//Cases to handle the automatic setup of the checker board
CASE caseState OF
	//Initialization of all the variables 
	000:
		IF (GVL.boardIsSetup = TRUE) THEN
			currentChecker :=0;
			currentStack := 0;
			currentStackPosition := 0;
			caseState := 010;
		END_IF
	//Moving Z axis up to start move to first stack	
	010:
		movePiece.zPos := zUp;
		caseState := 020;
	//Execute of the above move	
	020:
		movePiece.ExecuteMove := TRUE;
		caseState := 030;
	//Check to make sure above move finished
	030:
		IF (movePiece.MoveDone) THEN
			caseState := 190;
			movePiece.ExecuteMove := FALSE;
		END_IF
		
	//Input of the x and y coordinates of the stack that is currently getting picked from
	040:
		IF (currentStack < 3 ) THEN
			movePiece.xPos := xStackOffset + (xStackDistance * currentStack);
			movePiece.yPos := yStackOffset + (yStackDistance * currentStack);		
			movePiece.zPos := zUp;
			caseState := 050;
		END_IF
		
		IF (currentStack >=3 AND currentStack < 6 ) THEN
			movePiece.xPos := xStackOffset + (xStackDistance * currentStack);
			movePiece.yPos := yStackOffset + (yStackDistance * currentStack);		
			movePiece.zPos := zUp;
			caseState := 050;			
		END_IF
	//Execution of the move to the current stack being picked from	
	050:
		movePiece.ExecuteMove := TRUE;
		caseState := 060;
	//Check to make sure the execution of the move to the first stack was completed
	060:
		IF (movePiece.MoveDone) THEN
			caseState := 070;
			movePiece.ExecuteMove := FALSE;
		END_IF
	//Moving Z axis down to pick up the current checker and incrementing the stack position 
	070:
		movePiece.zPos := zDown - pieceOffset * ( 4 - currentStackPosition);
		currentStackPosition := currentStackPosition +1;
		IF (currentStackPosition = 5) THEN
			currentStackPosition := 0;
			currentStack := currentStack + 1;
			IF(currentStack = 2 OR currentStack = 5) THEN 
				currentStackPosition := 3;
			END_IF
		END_IF
		caseState := 080;
	//Execution of the z axis move downward to pick up current checker from current stack
	080:
		movePiece.ExecuteMove := TRUE;
		caseState := 090;
	//Check to make sure that the z axis move was properly executed, and closing of the gripper and delay to make sure that the gripper grabs the checker
	090:
		IF (movePiece.MoveDone) THEN
			caseState := 100;
			movePiece.ExecuteMove := FALSE;
			gripperMove := TRUE;
			wait.startTimer := TRUE;
		END_IF
	//Waiting for the timer to finish and then reinitializing it as false, as well as moving the z axis back up to move to the proper checker space
	100:
		IF (wait.done) THEN
			wait.startTimer := FALSE;
			gripperMove := FALSE;
			movePiece.zPos := zUp;
			caseState := 110;
		END_IF
	//Execution of the Z-axis move upwards to start move to proper board location 	
	110:
		movePiece.ExecuteMove := TRUE;
		caseState := 120;
	//Check to make sure that the above move is completed
	120: 
		IF (movePiece.MoveDone) THEN
			caseState := 130;
			movePiece.ExecuteMove := FALSE;
		END_IF
	//Input of x and y coordinates to proper checker board location depending on the color of the checker and the current check being placed
	130:
		IF (currentChecker < 12) THEN
			movePiece.xPos := xBoardOffset + (GVL.pieces[0,currentChecker].startingLocation[0] * spaceOffset); 
			movePiece.yPos := yboardOffset + (GVL.pieces[0,CurrentChecker].startingLocation[1] * spaceOffseT);
			currentChecker := currentChecker+1;
			caseState := 140;
		END_IF
		
		IF (currentChecker >= 12 AND currentChecker < 24) THEN
			movePiece.xPos := xBoardOffset + (GVL.pieces[1,currentChecker].startingLocation[0] *spaceOffset); 
			movePiece.yPos := yboardOffset + (GVL.pieces[1,CurrentChecker].startingLocation[1] *spaceOffseT);
			currentChecker := currentChecker+1;
			caseState :=140;
		END_IF
	//Execution of the above move to place checker on the proper board square	
	140:
		movePiece.ExecuteMove := TRUE;
		caseState := 150;
	//Check to make sure that the above move was completed	
	150:
		IF (movePiece.MoveDone) THEN;
			caseState := 160 ;
			movePiece.ExecuteMove := FALSE;
		END_IF
	//Move Z axis down to board level to prepare to drop it off	
	160:
		movePiece.zPos := zDown;
		caseState := 170;
	//Execution of the downward movement of the z axis to drop off the checker
	170:
		movePiece.ExecuteMove := TRUE;
		caseState := 180;
	//Check to make sure z axis moved, and opening the grippers to drop the current checker on the board square
	180:
		IF (movePiece.MoveDone) THEN
			caseState := 190;
			movePiece.ExecuteMove := FALSE;
			gripperMove := TRUE;
			wait.startTimer := TRUE;
		END_IF
	//Re-initializing the timer function and reseting the z axis above the board
	190:
		IF (wait.done) THEN
			wait.startTimer := FALSE;
			gripperMove := FALSE;
			movePiece.zPos := zUp;
			caseState := 020;
		END_IF
		
		IF (currentChecker = 23) THEN
			caseState := 200;
		END_IF
	//Case to hold program until the board is called to be reset
	200:
		IF (gameReset = TRUE) THEN
			caseState := 000;
		END_IF
END_CASE

movePiece(AxisGroup := XYZ);
wait();

END_PROGRAM

// CODESYS_SoftMotion_Win_V3/Application/GameplayFunctions/movePiece
FUNCTION movePiece : Piece
VAR_INPUT
	currentPiece : Piece;
	spaceX : INT; // space that you the user wants to move to
	spaceY : INT; // space that the user wants to move to
END_VAR
VAR
	spaceTranslation : ARRAY [0..1] OF INT; // small numbers (0-7) that indicate how many spaces a piece needs to be moved
	sizeOfMoveX : INT := 50;
	sizeOfMoveY : INT := -50;
END_VAR

// DOESN'T DO ANYTHING, DEPRECATE


IF(currentPiece.validMoveArr[spaceX, spaceY]) THEN
	
	// Tells you how many spaces you need to move
	spaceTranslation[0] := spaceX - currentPiece.currentLocation[0];
	spaceTranslation[1] := spaceY - currentPiece.currentLocation[1];

	// Converts spaces needed to move into pixels needed to move
	currentPiece.translatedLocation[0] := spaceTranslation[0] * sizeOfMoveX;
	currentPiece.translatedLocation[1] := spaceTranslation[1] * sizeOfMoveY;
	
	// sets old location to the current location
	currentPiece.oldLocation[0] := currentPiece.currentLocation[0];
	currentPiece.oldLocation[1] := currentPiece.currentLocation[1];
	
	// updates the current location
	currentPiece.currentLocation[0] := spaceX;
	currentPiece.currentLocation[1] := spaceY;
	
END_IF

movePiece := currentPiece;
currentPiece.isSelected := FALSE;

RETURN;

END_FUNCTION

// CODESYS_SoftMotion_Win_V3/Application/GameplayFunctions/HMISequence
PROGRAM HMISequence
VAR
END_VAR

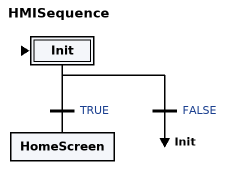
INITIAL_STEP Init:
END_STEP
TRANSITION FROM Init TO HomeScreen
    := TRUE;
END_TRANSITION
TRANSITION FROM Init TO Init
    := FALSE;
END_TRANSITION
STEP HomeScreen:
END_STEP

END_PROGRAM

// CODESYS_SoftMotion_Win_V3/Application/GameplayFunctions/Init
PROGRAM Init
VAR
END_VAR

END_PROGRAM

// CODESYS_SoftMotion_Win_V3/Application/GameplayFunctions/JumpPieces
PROGRAM JumpPieces
VAR
	i : INT;
	selectedPieceColor : INT;
	selectedPieceIndex : INT;
END_VAR

END_PROGRAM

// CODESYS_SoftMotion_Win_V3/Application/GameplayFunctions/pieceSelect
FUNCTION pieceSelect : ARRAY[0..1,0..11] OF Piece;
VAR_INPUT
	pieces : ARRAY[0..1,0..11] OF Piece;
	selectedPieceValidMoveArr : ARRAY[0..7,0..7] OF BOOL;
END_VAR
VAR
	i :INT;
END_VAR

FOR i := 0 TO 11 DO
	pieces[0,i].isSelected := FALSE;
	pieces[1,i].isSelected := FALSE;
END_FOR

selectedPieceValidMoveArr := pieces[0,10].validMoveArr;
pieceSelect := pieces;

END_FUNCTION

// CODESYS_SoftMotion_Win_V3/Application/GameplayFunctions/placePiece
FUNCTION placePiece : ARRAY [0..1] OF INT

VAR_INPUT
	isBlack : BOOL;
	pieceNum : INT;
END_VAR
VAR
	x : INT;
	y : INT;
	temp : INT;
END_VAR

// Set up for black
IF(isBlack) THEN
	y := pieceNum / 4;
	x := ((2 * pieceNum) MOD 8) + (y MOD 2);
// Setup for red
ELSE
	temp := pieceNum / 4;
	y := temp + 5;
	x := (((2 * pieceNum) MOD 8) + (temp MOD 2)) + 1;
	IF(x >= 8) THEN
		x := 0;
	END_IF
END_IF

placePiece[0] := x;
placePiece[1] := y;

RETURN;

END_FUNCTION

// CODESYS_SoftMotion_Win_V3/Application/GameplayFunctions/ProgramFlow
PROGRAM ProgramFlow
VAR
	PlayGame: BOOL;
END_VAR
// where we displace player move options?

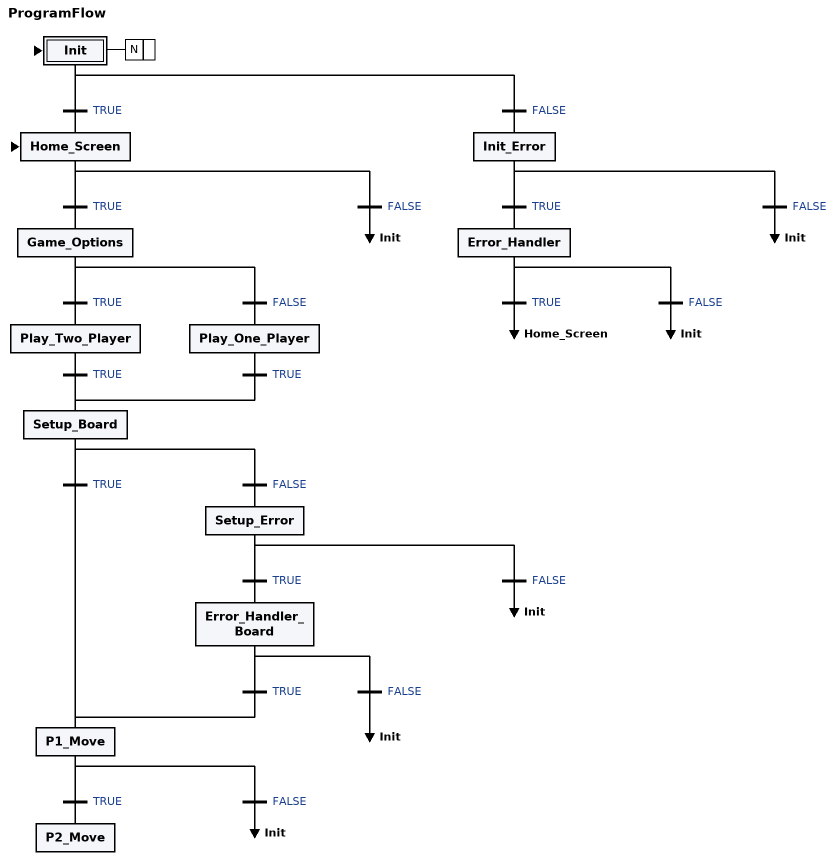
INITIAL_STEP Init:
    // ???(N);
END_STEP
TRANSITION FROM Init TO Home_Screen
    := TRUE;
END_TRANSITION
TRANSITION FROM Init TO Init_Error
    := FALSE;
END_TRANSITION
STEP Init_Error:
END_STEP
TRANSITION FROM Init_Error TO Error_Handler
    := TRUE;
END_TRANSITION
STEP Error_Handler:
END_STEP
TRANSITION FROM Error_Handler TO Home_Screen
    := TRUE;
END_TRANSITION
TRANSITION FROM Error_Handler TO Init
    := FALSE;
END_TRANSITION
TRANSITION FROM Init_Error TO Init
    := FALSE;
END_TRANSITION
STEP Home_Screen:
END_STEP
TRANSITION FROM Home_Screen TO Game_Options
    := TRUE;
END_TRANSITION
TRANSITION FROM Home_Screen TO Init
    := FALSE;
END_TRANSITION
STEP Game_Options:
END_STEP
TRANSITION FROM Game_Options TO Play_Two_Player
    := TRUE;
END_TRANSITION
STEP Play_Two_Player:
END_STEP
TRANSITION FROM Play_Two_Player TO Setup_Board
    := TRUE;
END_TRANSITION
TRANSITION FROM Game_Options TO Play_One_Player
    := FALSE;
END_TRANSITION
STEP Play_One_Player:
END_STEP
TRANSITION FROM Play_One_Player TO Setup_Board
    := TRUE;
END_TRANSITION
STEP Setup_Board:
END_STEP
TRANSITION FROM Setup_Board TO P1_Move
    := TRUE;
END_TRANSITION
TRANSITION FROM Setup_Board TO Setup_Error
    := FALSE;
END_TRANSITION
STEP Setup_Error:
END_STEP
TRANSITION FROM Setup_Error TO Error_Handler_Board
    := TRUE;
END_TRANSITION
TRANSITION FROM Setup_Error TO Init
    := FALSE;
END_TRANSITION
STEP Error_Handler_Board:
END_STEP
TRANSITION FROM Error_Handler_Board TO P1_Move
    := TRUE;
END_TRANSITION
TRANSITION FROM Error_Handler_Board TO Init
    := FALSE;
END_TRANSITION
STEP P1_Move:
END_STEP
TRANSITION FROM P1_Move TO P2_Move
    := TRUE;
END_TRANSITION
TRANSITION FROM P1_Move TO Init
    := FALSE;
END_TRANSITION
STEP P2_Move:
END_STEP

END_PROGRAM

// CODESYS_SoftMotion_Win_V3/Application/GameplayFunctions/MoveHome
PROGRAM MoveHome
VAR
	moveToHome : MovePieceMotion;
	caseState: INT;
END_VAR

CASE caseState OF
	
000: 
	IF(GVL.homeAxes)THEN
		moveToHome.xPos := 0;
		moveToHome.yPos := 0;
		moveToHome.zPos := 0;
		caseState := 010;
	END_IF

010:
	moveToHome.ExecuteMove := TRUE;
	caseState := 020;

020:
	IF(moveToHome.MoveDone)THEN
		moveToHome.ExecuteMove := FALSE;
		caseState := 000;
		GVL.homeAxes := FALSE;
	END_IF
	
	
END_CASE

moveToHome();

END_PROGRAM

// CODESYS_SoftMotion_Win_V3/Application/GameplayFunctions/SetupFromStart
PROGRAM SetupFromStart
VAR
END_VAR

END_PROGRAM

// CODESYS_SoftMotion_Win_V3/Application/ArrayMove
FUNCTION_BLOCK ArrayMove
VAR_INPUT
	//TestArray: ARRAY [1..20] OF INT := [1,2,3,4,5,6,7,8,9,10,11,12,13,14,15,16,17,18,19,20];
	i: INT ; 
END_VAR
VAR_OUTPUT
END_VAR
VAR
	Done : BOOL;
END_VAR

IF(NOT Done) THEN	
	FOR i:= 20 TO 2 BY -1 DO 
		PersistentVars.MyArray[i]:= PersistentVars.MyArray [i-1];
	END_FOR
	PersistentVars.MyArray[1].Names := GlobalVars.winnerName;
	PersistentVars.MyArray[1].Moves := GlobalVars.winnerMoves;
	Done := TRUE;
END_IF

END_FUNCTION_BLOCK

// CODESYS_SoftMotion_Win_V3/Application/GameplayFunctions/TestMyArray
PROGRAM TestMyArray
VAR
	k : INT ; 
	arrayTest : ArrayMove;
END_VAR

arrayTest();
//k := ArrayMove.TestArray[2];

END_PROGRAM

// CODESYS_SoftMotion_Win_V3/Application/Export/GetHeaderString
FUNCTION GetHeaderString : STRING[255]
VAR_INPUT
END_VAR
VAR
	msg: STRING[255];
	seperator: STRING;
	eol:String;
	strTemp0 : STRING[255];
	strTemp1 : STRING[255];
	

END_VAR

eol := WORD_AS_STRING(16#0A0D, FALSE);
seperator := ',';

strTemp0 := Concat(Concat(	'Winners', 
						 seperator), 
						    'Moves');




GetHeaderString := Concat(Concat(Concat(Concat(	'TimeStamp', 
														seperator),
														strTemp0), 
														seperator),
						     								eol);

END_FUNCTION

// CODESYS_SoftMotion_Win_V3/Application/Export/GetLogMsgString
FUNCTION GetLogMsgString : STRING[255]
VAR_INPUT
END_VAR
VAR
	msg: STRING[255];
	seperator: STRING;
	eol:String;
	
	DataPrep: STRING[255];
	
	
END_VAR

eol := WORD_AS_STRING(16#0A0D, FALSE);
seperator := ',';


DataPrep := Concat(Concat(  PersistentVars.MyArray[1].Names,
                                                  seperator),
            INT_TO_STRING(PersistentVars.MyArray[1].Moves));
																												



GetLogMsgString := Concat(Concat(Concat(Concat(	GetTimeStampString(),
														seperator),
														DataPrep), 
														seperator),
															eol);

END_FUNCTION

// CODESYS_SoftMotion_Win_V3/Application/Export/GetTimeStampString
FUNCTION GetTimeStampString : STRING
VAR_INPUT
END_VAR
VAR
	TimeStamp : SysTime;
	StructTimeStamp : SysTimeDate;
	Result : RTS_IEC_RESULT;
	StrDate : STRING;
	StrTime : STRING;
	

END_VAR

Result := systimertc.SysTimeRtcHighResGet(pTimestamp := TimeStamp);

Result := systimertc.SysTimeRtcConvertHighResToLocal(pTimeStamp:=TimeStamp, pDate:=StructTimeStamp);

StrDate := UINT_TO_STRING(StructTimeStamp.wYear);
IF StructTimeStamp.wMonth < 10 THEN 
	StrDate := Concat(Concat(StrDate, '0') , UINT_TO_STRING(StructTimeStamp.wMonth));
ELSE
	StrDate := Concat(StrDate , UINT_TO_STRING(StructTimeStamp.wMonth));
END_IF

IF StructTimeStamp.wDay < 10 THEN 
	StrDate := Concat(Concat(StrDate , '0') , UINT_TO_STRING(StructTimeStamp.wDay));
ELSE
	StrDate := Concat(StrDate , UINT_TO_STRING(StructTimeStamp.wDay));
END_IF


IF StructTimeStamp.wHour < 10 THEN 
	StrTime := Concat(Concat('0' , UINT_TO_STRING(StructTimeStamp.wHour)) , ':');
ELSE
	StrTime := Concat(UINT_TO_STRING(StructTimeStamp.wHour) , ':');
END_IF

IF StructTimeStamp.wMinute < 10 THEN 
	StrTime := Concat(Concat(Concat(StrTime , '0') , UINT_TO_STRING(StructTimeStamp.wMinute)), ':');
ELSE
	StrTime := Concat(Concat(StrTime , UINT_TO_STRING(StructTimeStamp.wMinute)), ':');
END_IF

IF StructTimeStamp.wSecond < 10 THEN 
	StrTime := Concat(Concat(Concat(StrTime , '0') , UINT_TO_STRING(StructTimeStamp.wSecond)) , '.');
ELSE
	StrTime := Concat(Concat(StrTime , UINT_TO_STRING(StructTimeStamp.wSecond)) , '.');
END_IF

IF StructTimeStamp.wMilliseconds < 10 THEN 
	StrTime := Concat(Concat(StrTime , '00') , UINT_TO_STRING(StructTimeStamp.wMilliseconds));
ELSE
	IF StructTimeStamp.wMilliseconds < 100 THEN 
		StrTime := Concat(Concat(StrTime , '0') , UINT_TO_STRING(StructTimeStamp.wMilliseconds));
	ELSE
		StrTime := Concat(StrTime , UINT_TO_STRING(StructTimeStamp.wMilliseconds));
	END_IF
END_IF

//GetTimeStampString := Concat(Concat(strDate , '-'), strTime);
GetTimeStampString := strTime;

END_FUNCTION

// CODESYS_SoftMotion_Win_V3/Application/Export/LogWinnerNames
PROGRAM LogWinnerNames
VAR
	strMsg: STRING[255];
	iStatus : INT := 0;
	LogIndex :DINT := 0;
	LogMsg : ARRAY [1..200] OF STRING[255];
	LogType : STRING;
	
	CycleTimeWarning: DWORD := 600;
	TotalSyncBufferAvgWarning: DINT := 125;
	CycleTimeError: DWORD := 900;
	TotalSyncBufferAvgError: DINT := 200;
	
	
	
END_VAR

VAR_INPUT
	bResetArray: BOOL;
END_VAR

IF bResetArray = TRUE THEN
	LogIndex := 0;
END_IF




CASE iStatus OF
	

0:	//Log Data
	LogIndex := LogIndex + 1;
	
	LogMsg[LogIndex] :=  GetLogMsgString();
	
	iStatus := 2;

END_CASE

END_PROGRAM

// CODESYS_SoftMotion_Win_V3/Application/Export/Run_FileCopy
PROGRAM Run_FileCopy
VAR
	RunTest: Test_FileCopy;
END_VAR

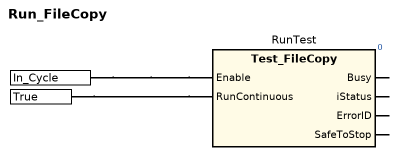
RunTest(Enable := In_Cycle, RunContinuous := True); // Test_FileCopy

END_PROGRAM

// CODESYS_SoftMotion_Win_V3/Application/Export/Test_FileCopy
FUNCTION_BLOCK Test_FileCopy
VAR_INPUT
	Enable: BOOL;
	RunContinuous:Bool := False;
END_VAR
VAR_OUTPUT
	Busy: BOOL;
	iStatus : INT := 0;
	ErrorID: INT;
	SafeToStop : Bool;
END_VAR
VAR
	OriginalFilePath : STRING := '/Hard disk/Backup/nk.bin';
	MemoryFilePath : STRING := '/nk.bin';
	USBFilePath : STRING := '/Hard disk2/nk.bin';
	DwellTime : TIME := T#15S;
	DoDwell : TON;
	
	Result1: SYSFILE.RTS_IEC_RESULT;
	Result2: SYSFILE.RTS_IEC_RESULT;

	BytesCopied: DWORD;
	SizeOriginal: DWORD;
	SizeMemory: DWORD;
	SizeUSB: DWORD;
END_VAR

IF Enable = FALSE and SafeToStop = True THEN
	iStatus := 0;
END_IF


CASE iStatus OF
	



0:  //Check Memory File Exist
	SafeToStop:=TRUE;
	SizeMemory := SysFileGetSize(MemoryFilePath, ADR(Result1));
	IF SizeMemory > 0 AND Result1 = Errors.ERR_OK THEN
		iStatus:=iStatus + 1;
	ELSE
		ErrorID := -1 * iStatus;  //Memory does not exist
		iStatus := 99;
	END_IF	

1:  //Check USB File Exist
	SafeToStop:=TRUE;
	SizeUSB := SysFileGetSize(USBFilePath, ADR(Result1));
	IF SizeUSB > 0 AND Result1 = Errors.ERR_OK THEN
		IF RunContinuous=TRUE THEN
			iStatus:=0;
		ELSE
			iStatus := 99;
		END_IF	
	ELSE
		ErrorID := -1 * iStatus;  //USB does not exist
		iStatus := 99;
	END_IF	
	
2:  // Copy to USBThumbdrive 
	SafeToStop:=FALSE;
	Result1:=SysFileCopy(USBFilePath,OriginalFilePath, ADR(BytesCopied));
	IF Result1=Errors.ERR_OK AND BytesCopied=SizeOriginal THEN
		iStatus:=iStatus + 1;
	ELSE
		ErrorID := -1 * iStatus;  //Copy to Memory Failed
		iStatus := 99;
	END_IF
	

3: //Got Error
	SafeToStop:=TRUE;
	Busy:=FALSE;
	
END_CASE

END_FUNCTION_BLOCK

// CODESYS_SoftMotion_Win_V3/Application/Visualizations/AreYouSure
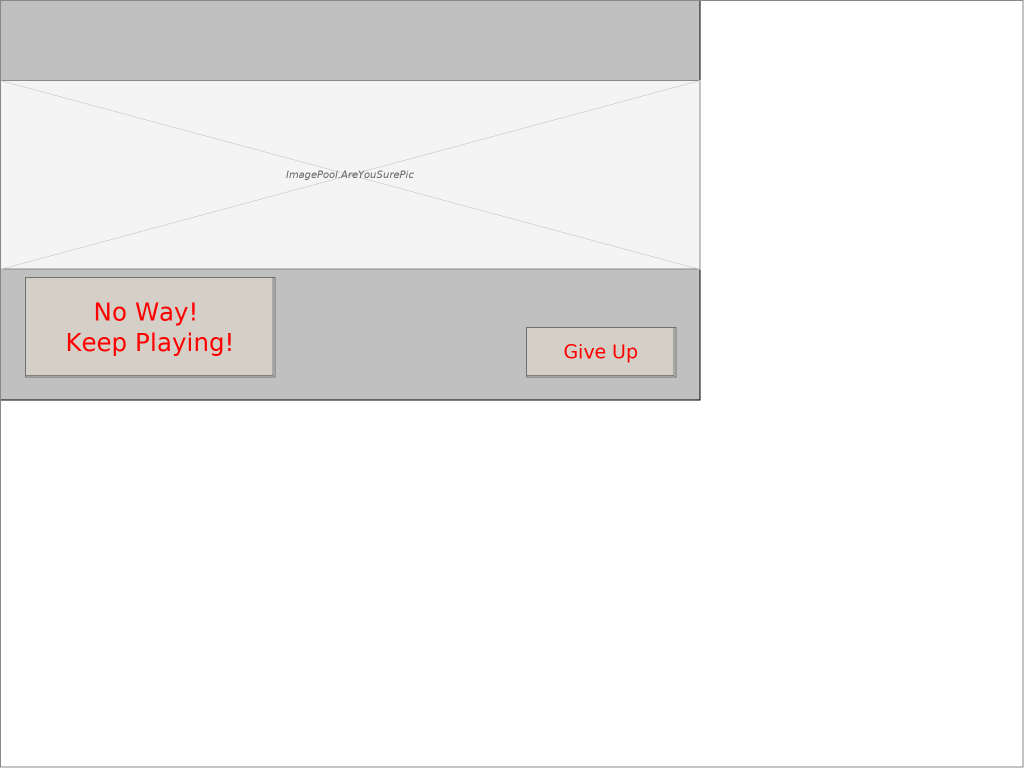
VISUALIZATION AreYouSure  // 1024x768
    Rectangle (0,0 700x400)
    Image (0,80 700x189), image: ImagePool.AreYouSurePic
    Button (25,277 250x100), "No Way! Keep Playing!"
        OnMouseClick:  Dialog=AreYouSure, Result=OK, NumpadKeypadSet=True
    Button (526,327 150x50), "Give Up"
        OnMouseClick:  Dialog=AreYouSure, Result=OK, NumpadKeypadSet=True
        OnMouseClick:  Assign=MainView, Type=Assignment
END_VISUALIZATION

// CODESYS_SoftMotion_Win_V3/Application/Visualizations/ErrorVis
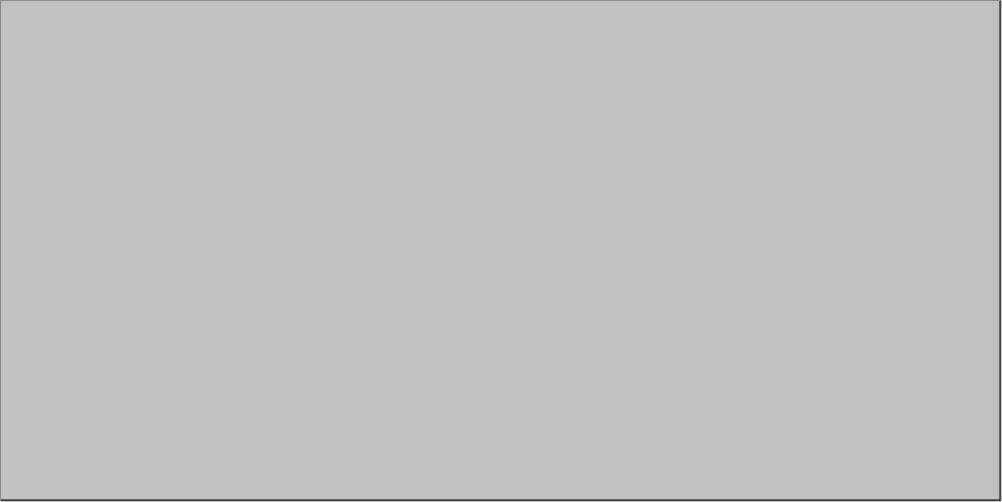
VISUALIZATION ErrorVis  // 1002x502
    Rectangle (0,0 1000x500)
END_VISUALIZATION

// CODESYS_SoftMotion_Win_V3/Application/Visualizations/JogVis
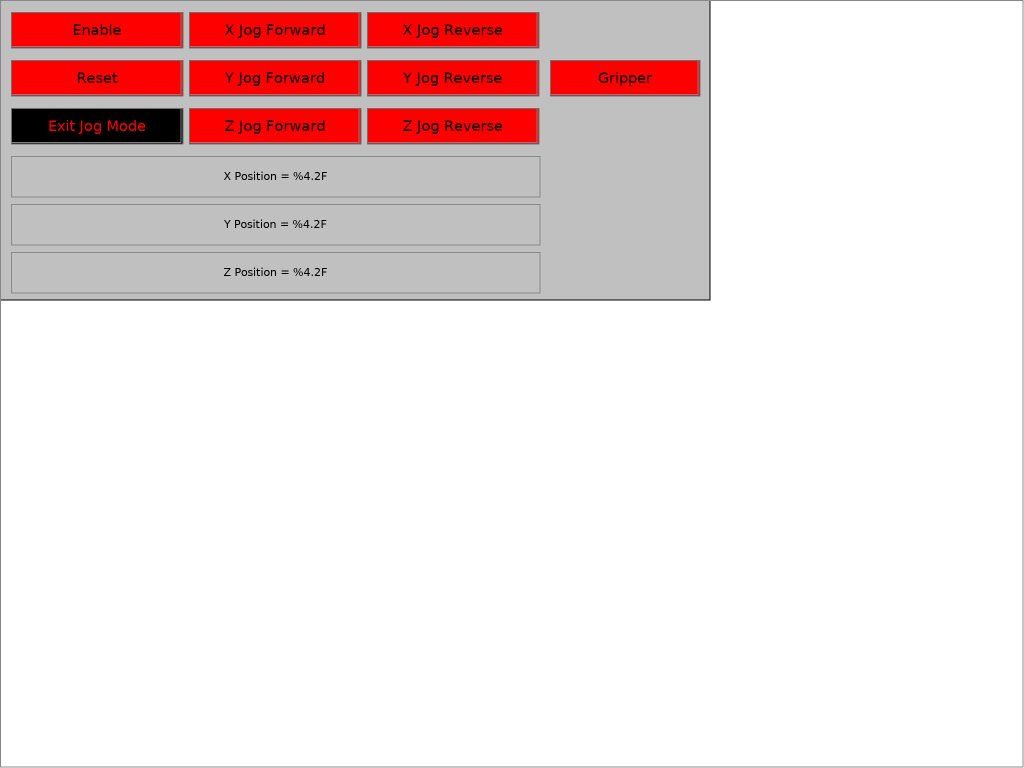
VISUALIZATION JogVis  // 1024x768
    Rectangle (0,0 710x300)
    Button (11,12 172x36), "Enable"
        OnMouseClick:  ToggleVariable=TestPower.Enable
        OnMouseClick: execute { GlobalVars.systemEnable := TRUE; }
    Button (189,12 172x36), "X Jog Forward"
        tap JogLogic.xJogFwdPressed
    Button (367,12 172x36), "X Jog Reverse"
        tap JogLogic.xJogRevPressed
    Button (189,60 172x36), "Y Jog Forward"
        tap JogLogic.yJogFwdPressed
    Button (367,60 172x36), "Y Jog Reverse"
        tap JogLogic.yJogRevPressed
    Button (11,60 172x36), "Reset"
        OnMouseClick: execute { TestPower.systemReset := TRUE; }
    Button (189,108 172x36), "Z Jog Forward"
        tap JogLogic.zJogFwdPressed
    Button (367,108 172x36), "Z Jog Reverse"
        tap JogLogic.zJogRevPressed
    Frame (11,156 529x41), "X Position = %4.2F", text variable: X.fActPosition
        shows SM3_Basic.LinDrive(m_Input_AXISREF := X)
    Frame (11,204 529x41), "Y Position = %4.2F", text variable: Y.fActPosition
        shows SM3_Basic.LinDrive(m_Input_AXISREF := Y)
    Frame (11,252 529x41), "Z Position = %4.2F", text variable: Z.fActPosition
        shows SM3_Basic.LinDrive(m_Input_AXISREF := Z)
    Button (11,108 172x36), "Exit Jog Mode"
        OnMouseClick:  Dialog=JogVis, Result=OK, NumpadKeypadSet=True
    Button (550,60 150x36), "Gripper"
        toggle GripperMove
END_VISUALIZATION

// CODESYS_SoftMotion_Win_V3/Application/Visualizations/GameView
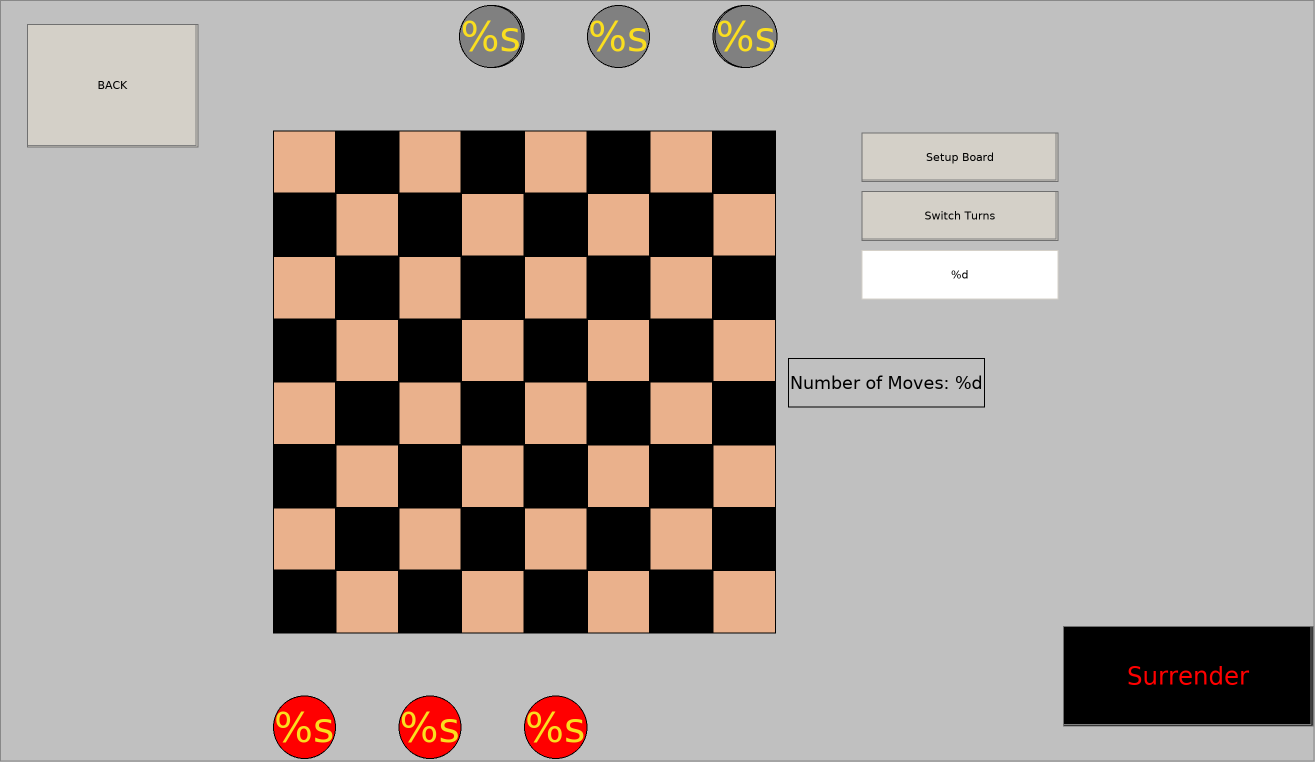
VISUALIZATION GameView  // 1315x762
    Frame (273,5 1005x755)
        shows Checkerboard()
    Button (27,24 171x123), "BACK"
        OnMouseClick:  Type=Previous
        OnMouseClick: execute { TestPower.GroupEnable := FALSE; }
    Button (1063,626 250x100), "Surrender"
        OnMouseClick:  Dialog=AreYouSure, OpenModal=True, OpenCentered=True
END_VISUALIZATION

// CODESYS_SoftMotion_Win_V3/Application/Visualizations/MainView
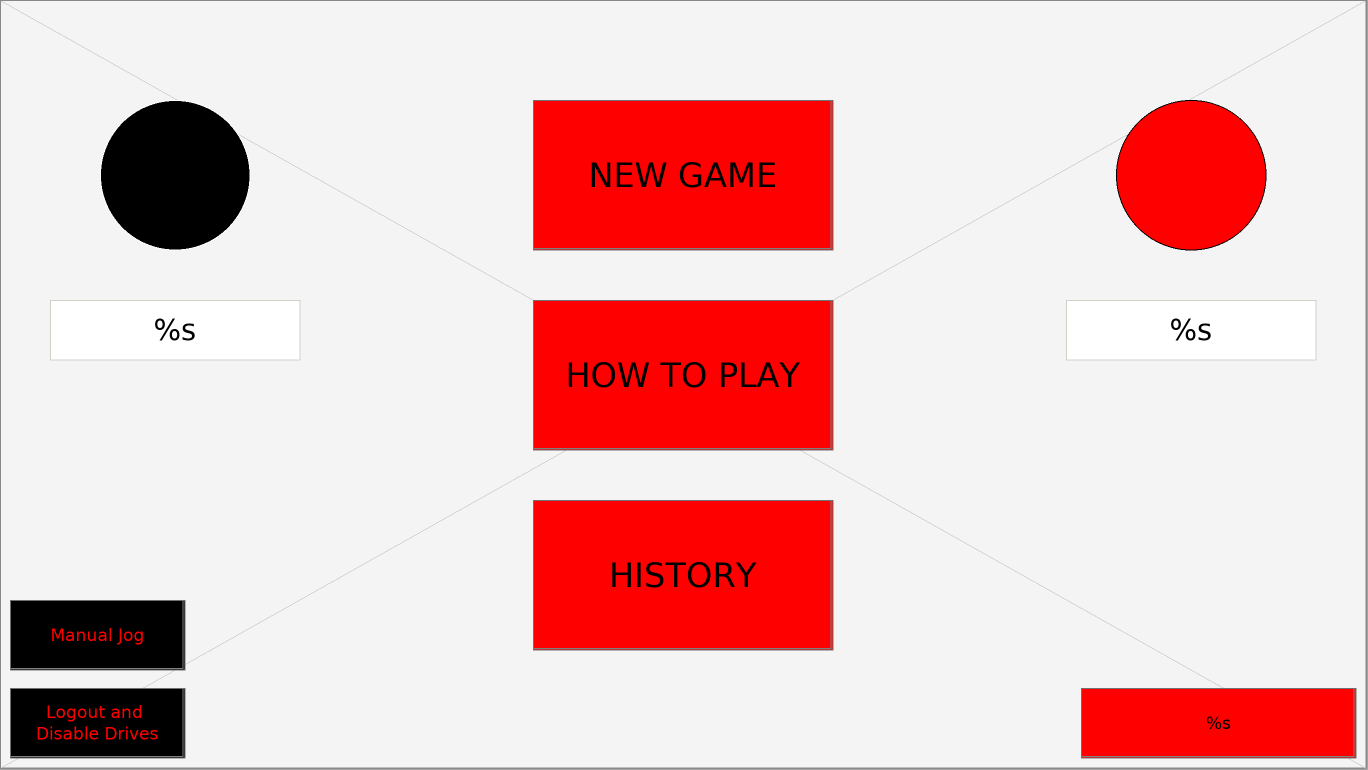
VISUALIZATION MainView  // 1368x770
    Image (0,0 1366x768), image: ImagePool.MedCheck_edited
    Ellipse (100,100 150x150), colour variable: GlobalVars.p1CheckerColor
    Ellipse (1116,100 150x150), colour variable: GlobalVars.p2CheckerColor
    Textfield (50,300 250x60), "%s", text variable: GlobalVars.p1Name
        OnMouseClick: write the text variable via Default
    Textfield (1066,300 250x60), "%s", text variable: GlobalVars.p2Name
        OnMouseClick: write the text variable via Default
    Button (533,100 300x150), "NEW GAME"
        OnMouseClick:  Assign=GameView, Type=Assignment
        OnMouseClick: execute { TestPower.GroupEnable := TRUE; }
    Button (533,300 300x150), "HOW TO PLAY"
        OnMouseClick:  Dialog=HowToPlay, OpenModal=True, OpenCentered=True
    Button (533,500 300x150), "HISTORY"
        OnMouseClick:  Dialog=History, OpenModal=True, OpenCentered=True
    Button (10,688 175x70), "Logout and Disable Drives"
        OnMouseClick:  Type=Logout
        OnMouseClick: execute { GlobalVars.systemEnable := FALSE; }
        OnMouseClick:  Assign=InitScreen, Type=Assignment
    Button (10,600 175x70), "Manual Jog"
        OnMouseClick:  Dialog=JogVis, OpenModal=True, OpenCentered=True, PositionX=0, PositionY=0
        OnMouseClick: execute { GlobalVars.systemEnable := TRUE; }
    Button (1081,688 275x70), "%s", text variable: GlobalVars.funnyText
        OnMouseClick: execute {
            GlobalVars.funnyCounter := GlobalVars.funnyCounter + 1;
            IF (GlobalVars.funnyCounter = 1) THEN
            	GlobalVars.funnyText := 'Stop it';
            ELSIF (GlobalVars.funnyCounter = 2) THEN
            	GlobalVars.funnyText := '.........';
            ELSIF (GlobalVars.funnyCounter = 3) THEN
            	GlobalVars.funnyText := 'How would you like it?';
            ELSIF (GlobalVars.funnyCounter = 4) THEN
            	GlobalVars.funnyText := 'Youre only wasting your time';
            ELSIF (GlobalVars.funnyCounter = 5) THEN
            	GlobalVars.funnyText := 'You win';
            ELSIF (GlobalVars.funnyCounter = 7) THEN
            	GlobalVars.funnyText := 'You dont give up easily';
            ELSIF (GlobalVars.funnyCounter = 8) THEN
            	GlobalVars.funnyText := 'Prize for your persistance';
            ELSIF (GlobalVars.funnyCounter = 9) THEN
            	GlobalVars.funnyText := 'lol';
            	VisuElems.CURRENTLANGUAGE := 'CowbellChinese';
            END_IF
        }
END_VISUALIZATION

// CODESYS_SoftMotion_Win_V3/Application/Visualizations/Congratulations
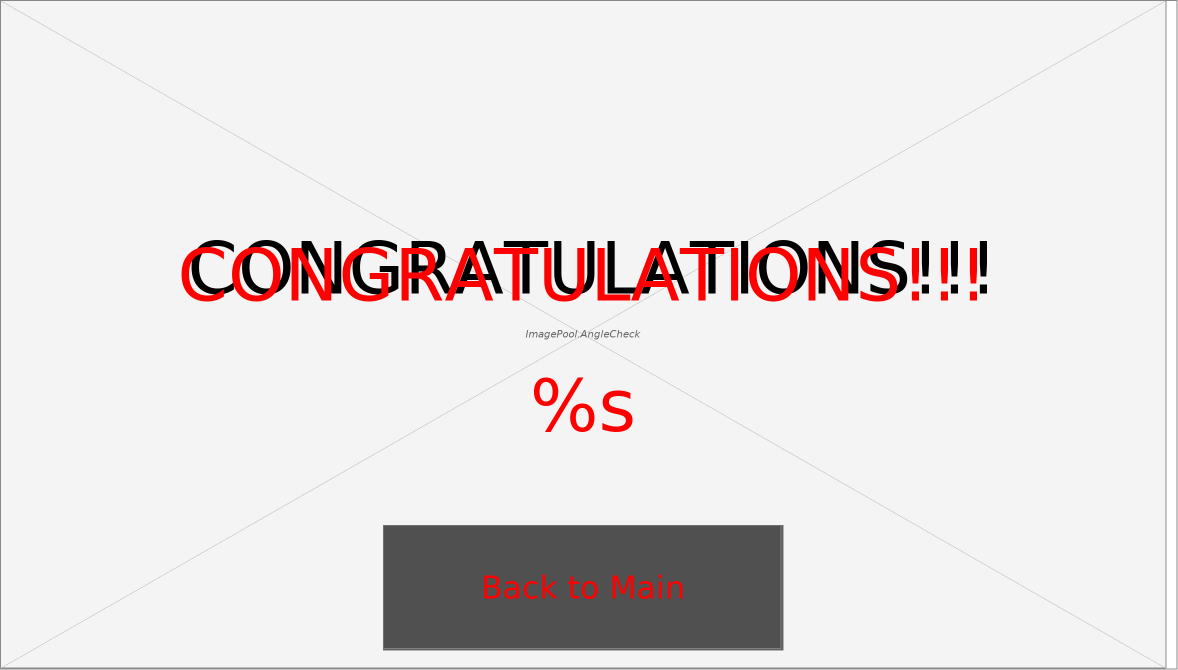
VISUALIZATION Congratulations  // 1178x670
    Image (0,0 1166x668), image: ImagePool.AngleCheck
    Rectangle (10,-7 1166x550), "CONGRATULATIONS!!!"
    Rectangle (0,0 1166x550), "CONGRATULATIONS!!!"
    Button (383,525 400x125), "Back to Main"
        OnMouseClick:  Assign=MainView, Type=Assignment
    Textfield (0,350 1166x111), "%s", text variable: GlobalVars.winnerName, colour variable: GlobalVars.p2CheckerColor
END_VISUALIZATION

// CODESYS_SoftMotion_Win_V3/Application/Visualizations/InitScreen
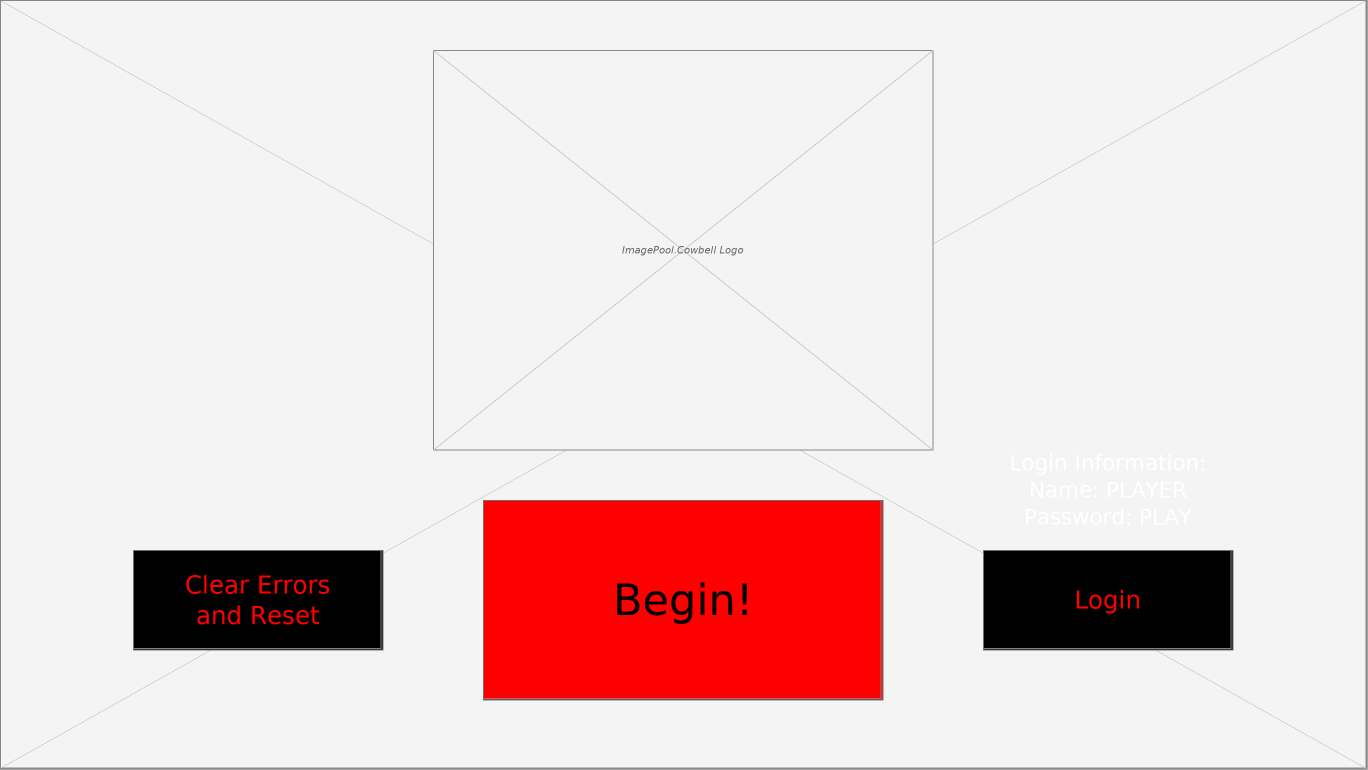
VISUALIZATION InitScreen  // 1368x770
    Image (0,0 1366x768), image: ImagePool.RedCheck
    Image (433,50 500x400), image: ImagePool.Cowbell Logo
    Button (483,500 400x200), "Begin!", text variable: GlobalVars.winnerName
        OnMouseClick:  Assign=MainView, Type=Assignment
        OnMouseClick: execute {
            TestPower.Enable := TRUE;
            JogLogic.startup := TRUE;
            // Run game setup code here
        }
    Button (983,550 250x100), "Login"
        OnMouseClick:  Type=Login
    Button (133,550 250x100), "Clear Errors and Reset"
        OnMouseClick: execute {
            VisuElems.CURRENTLANGUAGE := 'Default';
            JogLogic.startup := TRUE;
            // Any additional resets required to be done here
        }
        OnMouseClick:  Dialog=ErrorsCleared, OpenModal=True, OpenCentered=True
    Rectangle (983,440 250x100), "Login Information: Name: PLAYER Password: PLAY"
END_VISUALIZATION

// CODESYS_SoftMotion_Win_V3/Application/Visualizations/HowToPlay
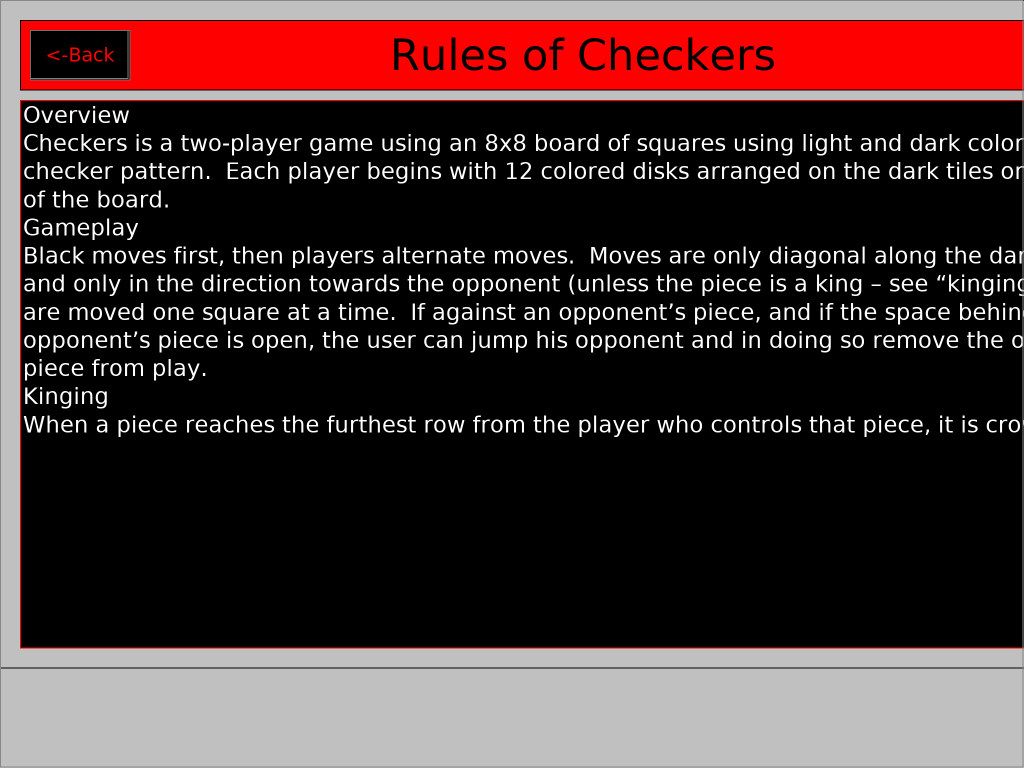
VISUALIZATION HowToPlay  // 1024x768
    Rectangle (0,0 1166x668)
    Textfield (20,100 1126x548), "Overview Checkers is a two-player game using an 8x8 board of squares using light and dark colors in a checker pattern. Each player begins with 12 colored disks arranged on the dark tiles on their side of the board. Gameplay Black moves first, then players alternate moves. Moves are only diagonal along the dark squares and only in the direction towards the opponent (unless the piece is a king – see “kinging”). Pieces are moved one square at a time. If against an opponent’s piece, and if the space behind the opponent’s piece is open, the user can jump his opponent and in doing so remove the opponent piece from play. Kinging When a piece reaches the furthest row from the player who controls that piece, it is crowned and becomes a king. One of the pieces which had been captured is placed on top of the king so that it is twice as high as a single piece. Kings may move both forward and backwards Winning A player wins the game when the opponent cannot make a move. In most cases, this is because all of the opponent's pieces have been captured, but it could also be because all of his pieces are blocked in."
    Textfield (20,20 1126x70), "Rules of Checkers"
    Button (30,30 100x50), "<-Back"
        OnMouseClick:  Dialog=HowToPlay, Result=OK, NumpadKeypadSet=True
END_VISUALIZATION

// CODESYS_SoftMotion_Win_V3/Application/Visualizations/ErrorsCleared
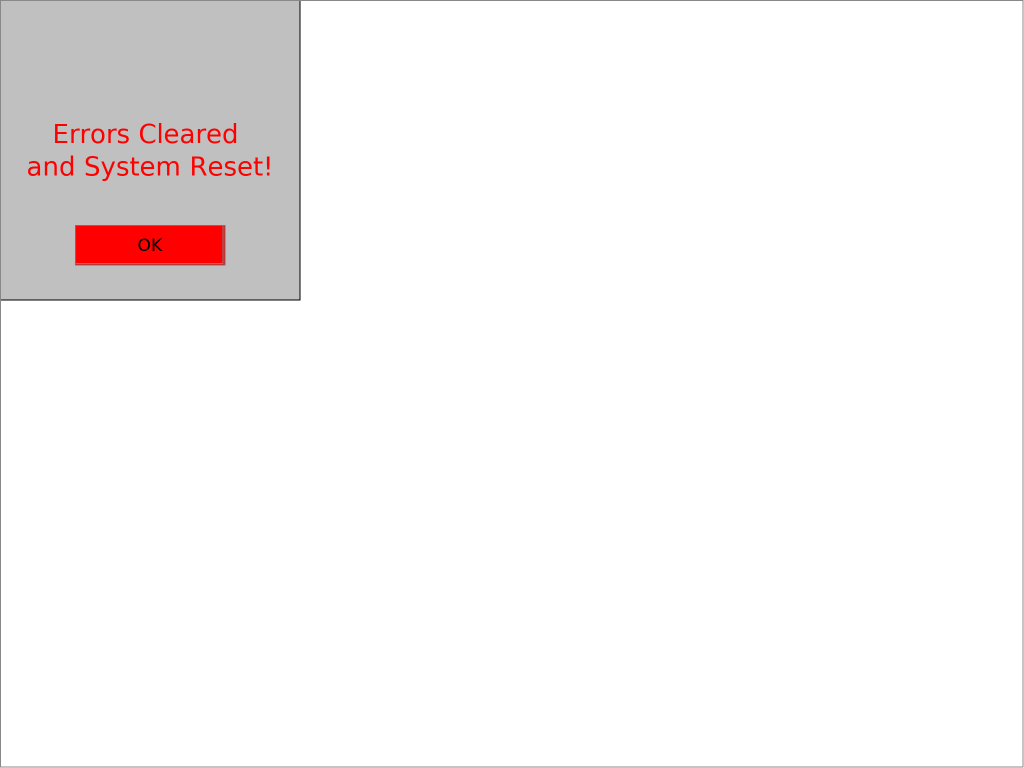
VISUALIZATION ErrorsCleared  // 1024x768
    Rectangle (0,0 300x300), "Errors Cleared and System Reset!"
    Button (75,225 150x40), "OK"
        OnMouseClick:  Dialog=ErrorsCleared, Result=OK, NumpadKeypadSet=True
END_VISUALIZATION

// CODESYS_SoftMotion_Win_V3/Application/Visualizations/Checkerboard
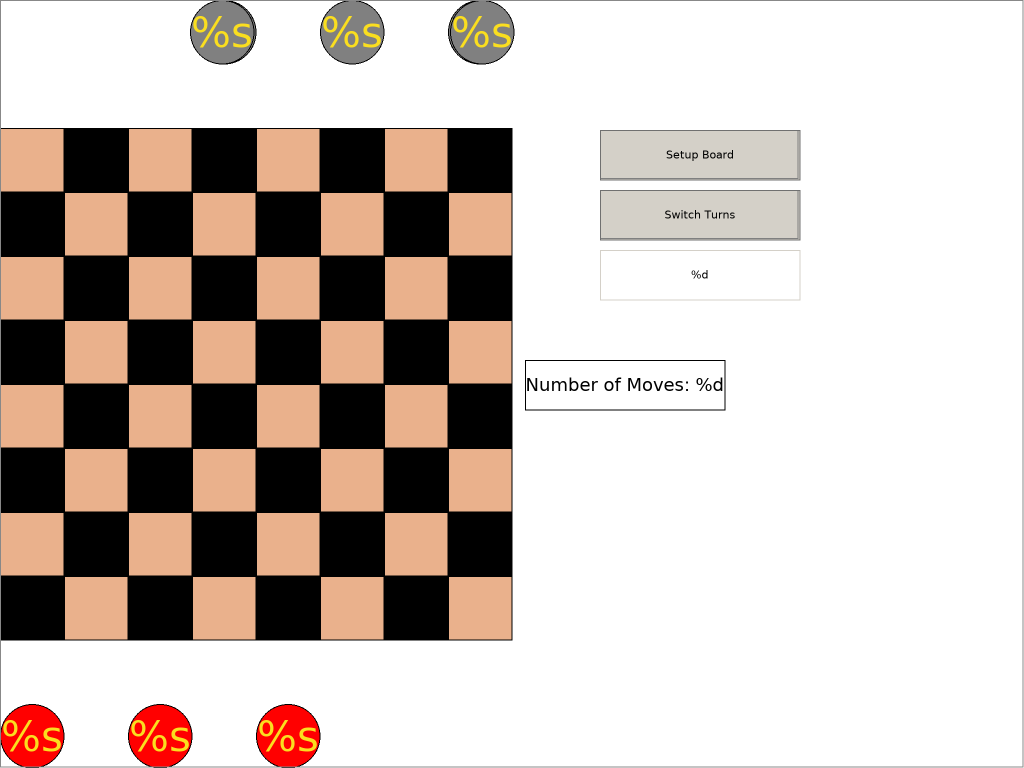
VISUALIZATION Checkerboard  // 1024x768
VAR_IN_OUT
	
END_VAR

VAR
	i : INT;
END_VAR
    Rectangle (0,320 64x64), colour toggle: GVL.selectedPieceValidMoveArr[0,4]
        OnMouseClick: execute { GVL.xMoveSpace := 0; GVL.yMoveSpace := 4; }
    Rectangle (64,320 64x64)
    Rectangle (128,320 64x64), colour toggle: GVL.selectedPieceValidMoveArr[2,4]
        OnMouseClick: execute { GVL.xMoveSpace := 2; GVL.yMoveSpace := 4; }
    Rectangle (192,320 64x64)
    Rectangle (0,256 64x64)
    Rectangle (64,256 64x64), colour toggle: GVL.selectedPieceValidMoveArr[1,5]
        OnMouseClick: execute { GVL.xMoveSpace := 1; GVL.yMoveSpace := 5; }
    Rectangle (128,256 64x64)
    Rectangle (192,256 64x64), colour toggle: GVL.selectedPieceValidMoveArr[3,5]
        OnMouseClick: execute { GVL.xMoveSpace := 3; GVL.yMoveSpace := 5; }
    Rectangle (0,192 64x64), colour toggle: GVL.selectedPieceValidMoveArr[0,6]
        OnMouseClick: execute { GVL.xMoveSpace := 0; GVL.yMoveSpace := 6; }
    Rectangle (64,192 64x64)
    Rectangle (128,192 64x64), colour toggle: GVL.selectedPieceValidMoveArr[2,6]
        OnMouseClick: execute { GVL.xMoveSpace := 2; GVL.yMoveSpace := 6; }
    Rectangle (192,192 64x64)
    Rectangle (0,128 64x64)
    Rectangle (192,128 64x64), colour toggle: GVL.selectedPieceValidMoveArr[3,7]
        OnMouseClick: execute { GVL.xMoveSpace := 3; GVL.yMoveSpace := 7; }
    Rectangle (128,128 64x64)
    Rectangle (64,128 64x64), colour toggle: GVL.selectedPieceValidMoveArr[1,7]
        OnMouseClick: execute { GVL.xMoveSpace := 1; GVL.yMoveSpace := 7; }
    Rectangle (256,320 64x64), colour toggle: GVL.selectedPieceValidMoveArr[4,4]
        OnMouseClick: execute { GVL.xMoveSpace := 4; GVL.yMoveSpace := 4; }
    Rectangle (320,320 64x64)
    Rectangle (384,320 64x64), colour toggle: GVL.selectedPieceValidMoveArr[6,4]
        OnMouseClick: execute { GVL.xMoveSpace := 6; GVL.yMoveSpace := 4; }
    Rectangle (448,320 64x64)
    Rectangle (256,256 64x64)
    Rectangle (320,256 64x64), colour toggle: GVL.selectedPieceValidMoveArr[5,5]
        OnMouseClick: execute { GVL.xMoveSpace := 5; GVL.yMoveSpace := 5; }
    Rectangle (384,256 64x64)
    Rectangle (448,256 64x64), colour toggle: GVL.selectedPieceValidMoveArr[7,5]
        OnMouseClick: execute { GVL.xMoveSpace := 7; GVL.yMoveSpace := 5; }
    Rectangle (256,192 64x64), colour toggle: GVL.selectedPieceValidMoveArr[4,6]
        OnMouseClick: execute { GVL.xMoveSpace := 4; GVL.yMoveSpace := 6; }
    Rectangle (320,192 64x64)
    Rectangle (384,192 64x64), colour toggle: GVL.selectedPieceValidMoveArr[6,6]
        OnMouseClick: execute { GVL.xMoveSpace := 6; GVL.yMoveSpace := 6; }
    Rectangle (448,192 64x64)
    Rectangle (256,128 64x64)
    Rectangle (448,128 64x64), colour toggle: GVL.selectedPieceValidMoveArr[7,7]
        OnMouseClick: execute { GVL.xMoveSpace := 7; GVL.yMoveSpace := 7; }
    Rectangle (384,128 64x64)
    Rectangle (320,128 64x64), colour toggle: GVL.selectedPieceValidMoveArr[5,7]
        OnMouseClick: execute { GVL.xMoveSpace := 5; GVL.yMoveSpace := 7; }
    Rectangle (256,576 64x64), colour toggle: GVL.selectedPieceValidMoveArr[4,0]
        OnMouseClick: execute { GVL.xMoveSpace := 4; GVL.yMoveSpace := 0; }
    Rectangle (320,576 64x64)
    Rectangle (384,576 64x64), colour toggle: GVL.selectedPieceValidMoveArr[6,0]
        OnMouseClick: execute { GVL.xMoveSpace := 6; GVL.yMoveSpace := 0; }
    Rectangle (448,576 64x64)
    Rectangle (256,512 64x64)
    Rectangle (320,512 64x64), colour toggle: GVL.selectedPieceValidMoveArr[5,1]
        OnMouseClick: execute { GVL.xMoveSpace := 5; GVL.yMoveSpace := 1; }
    Rectangle (384,512 64x64)
    Rectangle (448,512 64x64), colour toggle: GVL.selectedPieceValidMoveArr[7,1]
        OnMouseClick: execute { GVL.xMoveSpace := 7; GVL.yMoveSpace := 1; }
    Rectangle (256,448 64x64), colour toggle: GVL.selectedPieceValidMoveArr[4,2]
        OnMouseClick: execute { GVL.xMoveSpace := 4; GVL.yMoveSpace := 2; }
    Rectangle (320,448 64x64)
    Rectangle (384,448 64x64), colour toggle: GVL.selectedPieceValidMoveArr[6,2]
        OnMouseClick: execute { GVL.xMoveSpace := 6; GVL.yMoveSpace := 2; }
    Rectangle (448,448 64x64)
    Rectangle (256,384 64x64)
    Rectangle (448,384 64x64), colour toggle: GVL.selectedPieceValidMoveArr[7,3]
        OnMouseClick: execute { GVL.xMoveSpace := 7; GVL.yMoveSpace := 3; }
    Rectangle (384,384 64x64)
    Rectangle (320,384 64x64), colour toggle: GVL.selectedPieceValidMoveArr[5,3]
        OnMouseClick: execute { GVL.xMoveSpace := 5; GVL.yMoveSpace := 3; }
    Rectangle (0,576 64x64), colour toggle: GVL.selectedPieceValidMoveArr[0,0]
        OnMouseClick: execute { GVL.xMoveSpace := 0; GVL.yMoveSpace := 0; }
    Rectangle (64,576 64x64)
    Rectangle (128,576 64x64), colour toggle: GVL.selectedPieceValidMoveArr[2,0]
        OnMouseClick: execute { GVL.xMoveSpace := 2; GVL.yMoveSpace := 0; }
    Rectangle (192,576 64x64)
    Rectangle (0,512 64x64)
    Rectangle (64,512 64x64), colour toggle: GVL.selectedPieceValidMoveArr[1,1]
        OnMouseClick: execute { GVL.xMoveSpace := 1; GVL.yMoveSpace := 1; }
    Rectangle (128,512 64x64)
    Rectangle (192,512 64x64), colour toggle: GVL.selectedPieceValidMoveArr[3,1]
        OnMouseClick: execute { GVL.xMoveSpace := 3; GVL.yMoveSpace := 1; }
    Rectangle (0,448 64x64), colour toggle: GVL.selectedPieceValidMoveArr[0,2]
        OnMouseClick: execute { GVL.xMoveSpace := 0; GVL.yMoveSpace := 2; }
    Rectangle (64,448 64x64)
    Rectangle (128,448 64x64), colour toggle: GVL.selectedPieceValidMoveArr[2,2]
        OnMouseClick: execute { GVL.xMoveSpace := 2; GVL.yMoveSpace := 2; }
    Rectangle (192,448 64x64)
    Rectangle (0,384 64x64)
    Rectangle (192,384 64x64), colour toggle: GVL.selectedPieceValidMoveArr[3,3]
        OnMouseClick: execute { GVL.xMoveSpace := 3; GVL.yMoveSpace := 3; }
    Rectangle (128,384 64x64)
    Rectangle (64,384 64x64), colour toggle: GVL.selectedPieceValidMoveArr[1,3]
        OnMouseClick: execute { GVL.xMoveSpace := 1; GVL.yMoveSpace := 3; }
    Ellipse (256,704 64x64), "%s", text variable: GVL.pieces[0,11].kingText, colour toggle: GVL.pieces[0,11].isSelected
        p3560616238: GVL.pieces[0,11].translatedLocation[0]
        p2738717112: GVL.pieces[0,11].translatedLocation[1]
        OnMouseClick: execute {
            IF(NOT GVL.pieces[0,11].isSelected) THEN
            	// deselect everything
            	FOR i := 0 TO 11 DO
            		GVL.pieces[0,i].isSelected := FALSE;
            		GVL.pieces[1,i].isSelected := FALSE;
            	END_FOR
            	// select the piece
            	GVL.pieces[0,11].isSelected := TRUE;
            	GVL.selectedPieceValidMoveArr := GVL.pieces[0,11].validMoveArr;
            ELSE
            	GVL.pieces[0,11].isSelected := FALSE;
            	GVL.selectedPieceValidMoveArr := GVL.noValidMoveArr;
            END_IF
        }
    Ellipse (256,704 64x64), "%s", text variable: GVL.pieces[0,10].kingText, colour toggle: GVL.pieces[0,10].isSelected
        p3560616238: GVL.pieces[0,10].translatedLocation[0]
        p2738717112: GVL.pieces[0,10].translatedLocation[1]
        OnMouseClick: execute {
            IF(NOT GVL.pieces[0,10].isSelected) THEN
            	// deselect everything
            	FOR i := 0 TO 11 DO
            		GVL.pieces[0,i].isSelected := FALSE;
            		GVL.pieces[1,i].isSelected := FALSE;
            	END_FOR
            	// select the piece
            	GVL.pieces[0,10].isSelected := TRUE;
            	GVL.selectedPieceValidMoveArr := GVL.pieces[0,10].validMoveArr;
            ELSE
            	GVL.pieces[0,10].isSelected := FALSE;
            	GVL.selectedPieceValidMoveArr := GVL.noValidMoveArr;
            END_IF
        }
    Ellipse (128,704 64x64), "%s", text variable: GVL.pieces[0,9].kingText, colour toggle: GVL.pieces[0,9].isSelected
        p3560616238: GVL.pieces[0,9].translatedLocation[0]
        p2738717112: GVL.pieces[0,9].translatedLocation[1]
        OnMouseClick: execute {
            IF(NOT GVL.pieces[0,9].isSelected) THEN
            	// deselect everything
            	FOR i := 0 TO 11 DO
            		GVL.pieces[0,i].isSelected := FALSE;
            		GVL.pieces[1,i].isSelected := FALSE;
            	END_FOR
            	// select the piece
            	GVL.pieces[0,9].isSelected := TRUE;
            	GVL.selectedPieceValidMoveArr := GVL.pieces[0,9].validMoveArr;
            ELSE
            	GVL.pieces[0,9].isSelected := FALSE;
            	GVL.selectedPieceValidMoveArr := GVL.noValidMoveArr;
            END_IF
        }
    Ellipse (128,704 64x64), "%s", text variable: GVL.pieces[0,8].kingText, colour toggle: GVL.pieces[0,8].isSelected
        p3560616238: GVL.pieces[0,8].translatedLocation[0]
        p2738717112: GVL.pieces[0,8].translatedLocation[1]
        OnMouseClick: execute {
            IF(NOT GVL.pieces[0,8].isSelected) THEN
            	// deselect everything
            	FOR i := 0 TO 11 DO
            		GVL.pieces[0,i].isSelected := FALSE;
            		GVL.pieces[1,i].isSelected := FALSE;
            	END_FOR
            	// select the piece
            	GVL.pieces[0,8].isSelected := TRUE;
            	GVL.selectedPieceValidMoveArr := GVL.pieces[0,8].validMoveArr;
            ELSE
            	GVL.pieces[0,8].isSelected := FALSE;
            	GVL.selectedPieceValidMoveArr := GVL.noValidMoveArr;
            END_IF
        }
    Ellipse (128,704 64x64), "%s", text variable: GVL.pieces[0,7].kingText, colour toggle: GVL.pieces[0,7].isSelected
        p3560616238: GVL.pieces[0,7].translatedLocation[0]
        p2738717112: GVL.pieces[0,7].translatedLocation[1]
        OnMouseClick: execute {
            IF(NOT GVL.pieces[0,7].isSelected) THEN
            	// deselect everything
            	FOR i := 0 TO 11 DO
            		GVL.pieces[0,i].isSelected := FALSE;
            		GVL.pieces[1,i].isSelected := FALSE;
            	END_FOR
            	// select the piece
            	GVL.pieces[0,7].isSelected := TRUE;
            	GVL.selectedPieceValidMoveArr := GVL.pieces[0,7].validMoveArr;
            ELSE
            	GVL.pieces[0,7].isSelected := FALSE;
            	GVL.selectedPieceValidMoveArr := GVL.noValidMoveArr;
            END_IF
        }
    Ellipse (128,704 64x64), "%s", text variable: GVL.pieces[0,6].kingText, colour toggle: GVL.pieces[0,6].isSelected
        p3560616238: GVL.pieces[0,6].translatedLocation[0]
        p2738717112: GVL.pieces[0,6].translatedLocation[1]
        OnMouseClick: execute {
            IF(NOT GVL.pieces[0,6].isSelected) THEN
            	// deselect everything
            	FOR i := 0 TO 11 DO
            		GVL.pieces[0,i].isSelected := FALSE;
            		GVL.pieces[1,i].isSelected := FALSE;
            	END_FOR
            	// select the piece
            	GVL.pieces[0,6].isSelected := TRUE;
            	GVL.selectedPieceValidMoveArr := GVL.pieces[0,6].validMoveArr;
            ELSE
            	GVL.pieces[0,6].isSelected := FALSE;
            	GVL.selectedPieceValidMoveArr := GVL.noValidMoveArr;
            END_IF
        }
    Ellipse (128,704 64x64), "%s", text variable: GVL.pieces[0,5].kingText, colour toggle: GVL.pieces[0,5].isSelected
        p3560616238: GVL.pieces[0,5].translatedLocation[0]
        p2738717112: GVL.pieces[0,5].translatedLocation[1]
        OnMouseClick: execute {
            IF(NOT GVL.pieces[0,5].isSelected) THEN
            	// deselect everything
            	FOR i := 0 TO 11 DO
            		GVL.pieces[0,i].isSelected := FALSE;
            		GVL.pieces[1,i].isSelected := FALSE;
            	END_FOR
            	// select the piece
            	GVL.pieces[0,5].isSelected := TRUE;
            	GVL.selectedPieceValidMoveArr := GVL.pieces[0,5].validMoveArr;
            ELSE
            	GVL.pieces[0,5].isSelected := FALSE;
            	GVL.selectedPieceValidMoveArr := GVL.noValidMoveArr;
            END_IF
        }
    Ellipse (0,704 64x64), "%s", text variable: GVL.pieces[0,4].kingText, colour toggle: GVL.pieces[0,4].isSelected
        p3560616238: GVL.pieces[0,4].translatedLocation[0]
        p2738717112: GVL.pieces[0,4].translatedLocation[1]
        OnMouseClick: execute {
            IF(NOT GVL.pieces[0,4].isSelected) THEN
            	// deselect everything
            	FOR i := 0 TO 11 DO
            		GVL.pieces[0,i].isSelected := FALSE;
            		GVL.pieces[1,i].isSelected := FALSE;
            	END_FOR
            	// select the piece
            	GVL.pieces[0,4].isSelected := TRUE;
            	GVL.selectedPieceValidMoveArr := GVL.pieces[0,4].validMoveArr;
            ELSE
            	GVL.pieces[0,4].isSelected := FALSE;
            	GVL.selectedPieceValidMoveArr := GVL.noValidMoveArr;
            END_IF
        }
    Ellipse (0,704 64x64), "%s", text variable: GVL.pieces[0,3].kingText, colour toggle: GVL.pieces[0,3].isSelected
        p3560616238: GVL.pieces[0,3].translatedLocation[0]
        p2738717112: GVL.pieces[0,3].translatedLocation[1]
        OnMouseClick: execute {
            IF(NOT GVL.pieces[0,3].isSelected) THEN
            	// deselect everything
            	FOR i := 0 TO 11 DO
            		GVL.pieces[0,i].isSelected := FALSE;
            		GVL.pieces[1,i].isSelected := FALSE;
            	END_FOR
            	// select the piece
            	GVL.pieces[0,3].isSelected := TRUE;
            	GVL.selectedPieceValidMoveArr := GVL.pieces[0,3].validMoveArr;
            ELSE
            	GVL.pieces[0,3].isSelected := FALSE;
            	GVL.selectedPieceValidMoveArr := GVL.noValidMoveArr;
            END_IF
        }
    Ellipse (0,704 64x64), "%s", text variable: GVL.pieces[0,2].kingText, colour toggle: GVL.pieces[0,2].isSelected
        p3560616238: GVL.pieces[0,2].translatedLocation[0]
        p2738717112: GVL.pieces[0,2].translatedLocation[1]
        OnMouseClick: execute {
            IF(NOT GVL.pieces[0,2].isSelected) THEN
            	// deselect everything
            	FOR i := 0 TO 11 DO
            		GVL.pieces[0,i].isSelected := FALSE;
            		GVL.pieces[1,i].isSelected := FALSE;
            	END_FOR
            	// select the piece
            	GVL.pieces[0,2].isSelected := TRUE;
            	GVL.selectedPieceValidMoveArr := GVL.pieces[0,2].validMoveArr;
            ELSE
            	GVL.pieces[0,2].isSelected := FALSE;
            	GVL.selectedPieceValidMoveArr := GVL.noValidMoveArr;
            END_IF
        }
    Ellipse (0,704 64x64), "%s", text variable: GVL.pieces[0,1].kingText, colour toggle: GVL.pieces[0,1].isSelected
        p3560616238: GVL.pieces[0,1].translatedLocation[0]
        p2738717112: GVL.pieces[0,1].translatedLocation[1]
        OnMouseClick: execute {
            IF(NOT GVL.pieces[0,1].isSelected) THEN
            	// deselect everything
            	FOR i := 0 TO 11 DO
            		GVL.pieces[0,i].isSelected := FALSE;
            		GVL.pieces[1,i].isSelected := FALSE;
            	END_FOR
            	// select the piece
            	GVL.pieces[0,1].isSelected := TRUE;
            	GVL.selectedPieceValidMoveArr := GVL.pieces[0,1].validMoveArr;
            ELSE
            	GVL.pieces[0,1].isSelected := FALSE;
            	GVL.selectedPieceValidMoveArr := GVL.noValidMoveArr;
            END_IF
        }
    Ellipse (0,704 64x64), "%s", text variable: GVL.pieces[0,0].kingText, colour toggle: GVL.pieces[0,0].isSelected
        p3560616238: GVL.pieces[0,0].translatedLocation[0]
        p2738717112: GVL.pieces[0,0].translatedLocation[1]
        OnMouseClick: execute {
            IF(NOT GVL.pieces[0,0].isSelected) THEN
            	// deselect everything
            	FOR i := 0 TO 11 DO
            		GVL.pieces[0,i].isSelected := FALSE;
            		GVL.pieces[1,i].isSelected := FALSE;
            	END_FOR
            	// select the piece
            	GVL.pieces[0,0].isSelected := TRUE;
            	GVL.selectedPieceValidMoveArr := GVL.pieces[0,0].validMoveArr;
            ELSE
            	GVL.pieces[0,0].isSelected := FALSE;
            	GVL.selectedPieceValidMoveArr := GVL.noValidMoveArr;
            END_IF
        }
    Ellipse (192,0 64x64), "%s", text variable: GVL.pieces[1,11].kingText, colour toggle: GVL.pieces[1,11].isSelected
        p3560616238: GVL.pieces[1,11].translatedLocation[0]
        p2738717112: GVL.pieces[1,11].translatedLocation[1]
        OnMouseClick: execute {
            IF(NOT GVL.pieces[1,11].isSelected) THEN
            	// deselect everything
            	FOR i := 0 TO 11 DO
            		GVL.pieces[0,i].isSelected := FALSE;
            		GVL.pieces[1,i].isSelected := FALSE;
            	END_FOR
            	// select the piece
            	GVL.pieces[1,11].isSelected := TRUE;
            	GVL.selectedPieceValidMoveArr := GVL.pieces[1,11].validMoveArr;
            ELSE
            	GVL.pieces[1,11].isSelected := FALSE;
            	GVL.selectedPieceValidMoveArr := GVL.noValidMoveArr;
            END_IF
        }
    Ellipse (190,0 64x64), "%s", text variable: GVL.pieces[1,10].kingText, colour toggle: GVL.pieces[1,10].isSelected
        p3560616238: GVL.pieces[1,10].translatedLocation[0]
        p2738717112: GVL.pieces[1,10].translatedLocation[1]
        OnMouseClick: execute {
            IF(NOT GVL.pieces[1,10].isSelected) THEN
            	// deselect everything
            	FOR i := 0 TO 11 DO
            		GVL.pieces[0,i].isSelected := FALSE;
            		GVL.pieces[1,i].isSelected := FALSE;
            	END_FOR
            	// select the piece
            	GVL.pieces[1,10].isSelected := TRUE;
            	GVL.selectedPieceValidMoveArr := GVL.pieces[1,10].validMoveArr;
            ELSE
            	GVL.pieces[1,10].isSelected := FALSE;
            	GVL.selectedPieceValidMoveArr := GVL.noValidMoveArr;
            END_IF
        }
    Ellipse (320,0 64x64), "%s", text variable: GVL.pieces[1,9].kingText, colour toggle: GVL.pieces[1,9].isSelected
        p3560616238: GVL.pieces[1,9].translatedLocation[0]
        p2738717112: GVL.pieces[1,9].translatedLocation[1]
        OnMouseClick: execute {
            IF(NOT GVL.pieces[1,9].isSelected) THEN
            	// deselect everything
            	FOR i := 0 TO 11 DO
            		GVL.pieces[0,i].isSelected := FALSE;
            		GVL.pieces[1,i].isSelected := FALSE;
            	END_FOR
            	// select the piece
            	GVL.pieces[1,9].isSelected := TRUE;
            	GVL.selectedPieceValidMoveArr := GVL.pieces[1,9].validMoveArr;
            ELSE
            	GVL.pieces[1,9].isSelected := FALSE;
            	GVL.selectedPieceValidMoveArr := GVL.noValidMoveArr;
            END_IF
        }
    Ellipse (320,0 64x64), "%s", text variable: GVL.pieces[1,8].kingText, colour toggle: GVL.pieces[1,8].isSelected
        p3560616238: GVL.pieces[1,8].translatedLocation[0]
        p2738717112: GVL.pieces[1,8].translatedLocation[1]
        OnMouseClick: execute {
            IF(NOT GVL.pieces[1,8].isSelected) THEN
            	// deselect everything
            	FOR i := 0 TO 11 DO
            		GVL.pieces[0,i].isSelected := FALSE;
            		GVL.pieces[1,i].isSelected := FALSE;
            	END_FOR
            	// select the piece
            	GVL.pieces[1,8].isSelected := TRUE;
            	GVL.selectedPieceValidMoveArr := GVL.pieces[1,8].validMoveArr;
            ELSE
            	GVL.pieces[1,8].isSelected := FALSE;
            	GVL.selectedPieceValidMoveArr := GVL.noValidMoveArr;
            END_IF
        }
    Ellipse (320,0 64x64), "%s", text variable: GVL.pieces[1,7].kingText, colour toggle: GVL.pieces[1,7].isSelected
        p3560616238: GVL.pieces[1,7].translatedLocation[0]
        p2738717112: GVL.pieces[1,7].translatedLocation[1]
        OnMouseClick: execute {
            IF(NOT GVL.pieces[1,7].isSelected) THEN
            	// deselect everything
            	FOR i := 0 TO 11 DO
            		GVL.pieces[0,i].isSelected := FALSE;
            		GVL.pieces[1,i].isSelected := FALSE;
            	END_FOR
            	// select the piece
            	GVL.pieces[1,7].isSelected := TRUE;
            	GVL.selectedPieceValidMoveArr := GVL.pieces[1,7].validMoveArr;
            ELSE
            	GVL.pieces[1,7].isSelected := FALSE;
            	GVL.selectedPieceValidMoveArr := GVL.noValidMoveArr;
            END_IF
        }
    Ellipse (320,0 64x64), "%s", text variable: GVL.pieces[1,6].kingText, colour toggle: GVL.pieces[1,6].isSelected
        p3560616238: GVL.pieces[1,6].translatedLocation[0]
        p2738717112: GVL.pieces[1,6].translatedLocation[1]
        OnMouseClick: execute {
            IF(NOT GVL.pieces[1,6].isSelected) THEN
            	// deselect everything
            	FOR i := 0 TO 11 DO
            		GVL.pieces[0,i].isSelected := FALSE;
            		GVL.pieces[1,i].isSelected := FALSE;
            	END_FOR
            	// select the piece
            	GVL.pieces[1,6].isSelected := TRUE;
            	GVL.selectedPieceValidMoveArr := GVL.pieces[1,6].validMoveArr;
            ELSE
            	GVL.pieces[1,6].isSelected := FALSE;
            	GVL.selectedPieceValidMoveArr := GVL.noValidMoveArr;
            END_IF
        }
    Ellipse (320,0 64x64), "%s", text variable: GVL.pieces[1,5].kingText, colour toggle: GVL.pieces[1,5].isSelected
        p3560616238: GVL.pieces[1,5].translatedLocation[0]
        p2738717112: GVL.pieces[1,5].translatedLocation[1]
        OnMouseClick: execute {
            IF(NOT GVL.pieces[1,5].isSelected) THEN
            	// deselect everything
            	FOR i := 0 TO 11 DO
            		GVL.pieces[0,i].isSelected := FALSE;
            		GVL.pieces[1,i].isSelected := FALSE;
            	END_FOR
            	// select the piece
            	GVL.pieces[1,5].isSelected := TRUE;
            	GVL.selectedPieceValidMoveArr := GVL.pieces[1,5].validMoveArr;
            ELSE
            	GVL.pieces[1,5].isSelected := FALSE;
            	GVL.selectedPieceValidMoveArr := GVL.noValidMoveArr;
            END_IF
        }
    Ellipse (448,0 64x64), "%s", text variable: GVL.pieces[1,4].kingText, colour toggle: GVL.pieces[1,4].isSelected
        p3560616238: GVL.pieces[1,4].translatedLocation[0]
        p2738717112: GVL.pieces[1,4].translatedLocation[1]
        OnMouseClick: execute {
            IF(NOT GVL.pieces[1,4].isSelected) THEN
            	// deselect everything
            	FOR i := 0 TO 11 DO
            		GVL.pieces[0,i].isSelected := FALSE;
            		GVL.pieces[1,i].isSelected := FALSE;
            	END_FOR
            	// select the piece
            	GVL.pieces[1,4].isSelected := TRUE;
            	GVL.selectedPieceValidMoveArr := GVL.pieces[1,4].validMoveArr;
            ELSE
            	GVL.pieces[1,4].isSelected := FALSE;
            	GVL.selectedPieceValidMoveArr := GVL.noValidMoveArr;
            END_IF
        }
    Ellipse (450,0 64x64), "%s", text variable: GVL.pieces[1,3].kingText, colour toggle: GVL.pieces[1,3].isSelected
        p3560616238: GVL.pieces[1,3].translatedLocation[0]
        p2738717112: GVL.pieces[1,3].translatedLocation[1]
        OnMouseClick: execute {
            IF(NOT GVL.pieces[1,3].isSelected) THEN
            	// deselect everything
            	FOR i := 0 TO 11 DO
            		GVL.pieces[0,i].isSelected := FALSE;
            		GVL.pieces[1,i].isSelected := FALSE;
            	END_FOR
            	// select the piece
            	GVL.pieces[1,3].isSelected := TRUE;
            	GVL.selectedPieceValidMoveArr := GVL.pieces[1,3].validMoveArr;
            ELSE
            	GVL.pieces[1,3].isSelected := FALSE;
            	GVL.selectedPieceValidMoveArr := GVL.noValidMoveArr;
            END_IF
        }
    Ellipse (450,0 64x64), "%s", text variable: GVL.pieces[1,2].kingText, colour toggle: GVL.pieces[1,2].isSelected
        p3560616238: GVL.pieces[1,2].translatedLocation[0]
        p2738717112: GVL.pieces[1,2].translatedLocation[1]
        OnMouseClick: execute {
            IF(NOT GVL.pieces[1,2].isSelected) THEN
            	// deselect everything
            	FOR i := 0 TO 11 DO
            		GVL.pieces[0,i].isSelected := FALSE;
            		GVL.pieces[1,i].isSelected := FALSE;
            	END_FOR
            	// select the piece
            	GVL.pieces[1,2].isSelected := TRUE;
            	GVL.selectedPieceValidMoveArr := GVL.pieces[1,2].validMoveArr;
            ELSE
            	GVL.pieces[1,2].isSelected := FALSE;
            	GVL.selectedPieceValidMoveArr := GVL.noValidMoveArr;
            END_IF
        }
    Ellipse (450,0 64x64), "%s", text variable: GVL.pieces[1,1].kingText, colour toggle: GVL.pieces[1,1].isSelected
        p3560616238: GVL.pieces[1,1].translatedLocation[0]
        p2738717112: GVL.pieces[1,1].translatedLocation[1]
        OnMouseClick: execute {
            IF(NOT GVL.pieces[1,1].isSelected) THEN
            	// deselect everything
            	FOR i := 0 TO 11 DO
            		GVL.pieces[0,i].isSelected := FALSE;
            		GVL.pieces[1,i].isSelected := FALSE;
            	END_FOR
            	// select the piece
            	GVL.pieces[1,1].isSelected := TRUE;
            	GVL.selectedPieceValidMoveArr := GVL.pieces[1,1].validMoveArr;
            ELSE
            	GVL.pieces[1,1].isSelected := FALSE;
            	GVL.selectedPieceValidMoveArr := GVL.noValidMoveArr;
            END_IF
        }
    Ellipse (450,0 64x64), "%s", text variable: GVL.pieces[1,0].kingText, colour toggle: GVL.pieces[1,0].isSelected
        p3560616238: GVL.pieces[1,0].translatedLocation[0]
        p2738717112: GVL.pieces[1,0].translatedLocation[1]
        OnMouseClick: execute {
            IF(NOT GVL.pieces[1,0].isSelected) THEN
            	// deselect everything
            	FOR i := 0 TO 11 DO
            		GVL.pieces[0,i].isSelected := FALSE;
            		GVL.pieces[1,i].isSelected := FALSE;
            	END_FOR
            	// select the piece
            	GVL.pieces[1,0].isSelected := TRUE;
            	GVL.selectedPieceValidMoveArr := GVL.pieces[1,0].validMoveArr;
            ELSE
            	GVL.pieces[1,0].isSelected := FALSE;
            	GVL.selectedPieceValidMoveArr := GVL.noValidMoveArr;
            END_IF
        }
    Button (600,130 200x50), "Setup Board"
        tap Gameplay.commenceSetup
    Button (600,190 200x50), "Switch Turns"
        OnMouseClick:  ToggleVariable=GVL.redsTurn
    Textfield (600,250 200x50), "%d", text variable: GVL.blackPiecesTaken
    Rectangle (525,360 200x50), "Number of Moves: %d", text variable: GlobalVars.winnerMoves
END_VISUALIZATION

// CODESYS_SoftMotion_Win_V3/Application/MobileVisualizations/MobileVis
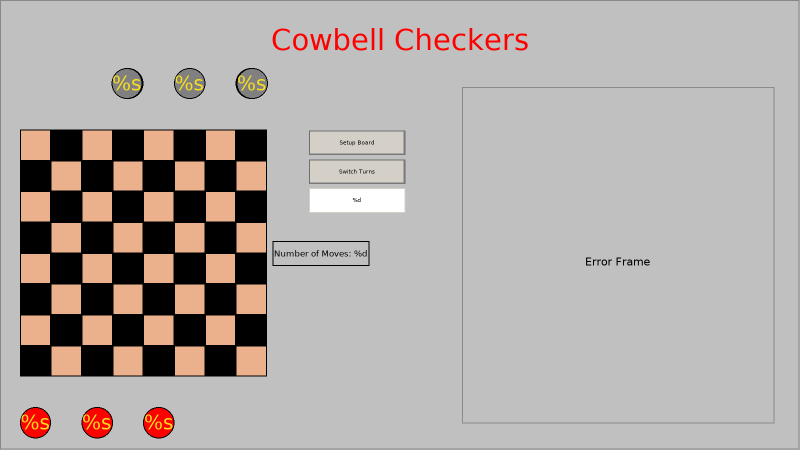
VISUALIZATION MobileVis  // 800x450
    Rectangle (250,15 300x50), "Cowbell Checkers"
    Frame (20,68 651x370)
        shows Checkerboard()
    Frame (462,87 312x336), "Error Frame"
END_VISUALIZATION

// CODESYS_SoftMotion_Win_V3/Application/Visualizations/History
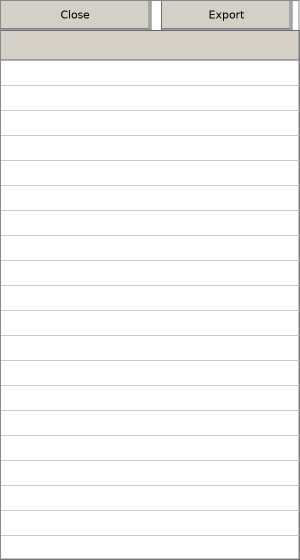
VISUALIZATION History  // 300x560
    Table (0,30 300x530), data array: PersistentVars.MyArray
        p3854506369: PersistentVars.MyArray[INDEX].Names
        p1892666644: PersistentVars.MyArray[INDEX].Moves
        p2232123230: Winners
    Button (0,0 151x30), "Close"
        OnMouseClick:  Dialog=History, Result=OK, NumpadKeypadSet=True
    Button (161,0 131x30), "Export"
        OnMouseClick: execute { GVL.export := TRUE; }
END_VISUALIZATION

(* text COWBELL_PROGRAMMING_STANDARD
*** General Team Guidelines ***

Program Names (Func, FB, Prog): ProgramName, Program_Name
-Which ever way appears more readable

Variable Names: var1, xVelocity, yVel1
-If global axis variable, axis identifier leads descriptive name.  start lowercase, camelCase

Functions, FunctionBlocks: These should not use global variables, if it can be avoided.  
These types should be able to copy and paste into a new program.

( * Header Comment * ) - good for describing chuncks of code
// In line comment - good for describing a single line

Programs, GlobalVars, etc. will be placed in the POUs so that we can work with the simulator from home.  Don't forget to copy programs to the required task!


Functions can only be called, take inputs and have defined outputs.  Good for math or modifiers.
Function Blocks must be called in a program and do not have explicitly defined inputs and outputs.  Good for repetive chunks of code.  
Programs are the only items that are run in the Task Configuration list.  Programs will call Functions and Function Blocks as required.  

*For Visual Stuff, let's try to stay with the Arial family of Fonts
*)

(* text GameInformation
Logins:

Admin : 1234
Tech : 123
User: play
*)
